FUNCTION_BLOCK FB_StateMachine
VAR_INPUT
	bStart: BOOL;
	bStop: BOOL;
END_VAR
VAR_OUTPUT
	Green: BOOL;
	Yellow: BOOL;
	Red: BOOL;
END_VAR
VAR
	State: E_States;
	T_Green: TON;
	T_Yellow: TON;
	T_Red: TON;
END_VAR

IF (bStop) THEN
	State:= E_States.eStop;
	//Reset dei timer
	T_Green(IN:= FALSE);
	T_Yellow(IN:= FALSE);
	T_Red(IN:= FALSE);
END_IF

CASE State OF
	E_States.eStop:
		Green:= FALSE;
		Yellow:= FALSE;
		Red:= FALSE;
		IF (NOT bStop AND bSTart) THEN
			State := E_States.eGreen; //Passo allo stato Verde
		END_IF
	
	E_States.eGreen:
		T_Green(IN:= TRUE, PT:= T#5S);
		Green:= TRUE;
		Yellow:= FALSE;
		Red:= FALSE;
		IF (T_Green.Q) THEN //Il tempo del verde è scaduto
			T_Green(IN:= FALSE); //Reset del timer verde 
			State := E_States.eYellow; //Passo allo stato Giallo
		END_IF

	E_States.eYellow:
		T_Yellow(IN:= TRUE, PT:= T#2S);
		Green:= TRUE;
		Yellow:= TRUE;
		Red:= FALSE;
		IF (T_Yellow.Q) THEN //Il tempo del giallo è scaduto
			T_Yellow(IN:= FALSE); //Reset del timer giallo 
			State := E_States.eRed; //Passo allo stato Rosso
		END_IF
		
	E_States.eRed:
		T_Red(IN:= TRUE, PT:= T#8S);
		Green:= FALSE;
		Yellow:= FALSE;
		Red:= TRUE;
		IF (T_Red.Q) THEN //Il tempo del rosso è scaduto
			T_Red(IN:= FALSE); //Reset del timer rosso 
			State := E_States.eGreen; //Passo allo stato Verde
		END_IF
	
END_CASE

END_FUNCTION_BLOCK

(* stored: Version 1.1.0.1, ProductVersion 3.1.4024.12
   POU FB_StateMachine: Id {f0fdb729-a96a-4ef9-9b71-68fec912dd01}, SpecialFunc None *)
